{attribute 'qualified_only'}
VAR_GLOBAL
		Device_1_EtherCAT : Device_1_EtherCAT_9EEE92A7;
END_VAR

(* stored: Version 1.2.0.0, ProductVersion 3.1.4024.11
   GVL GVL_iXlinker: Id {c7a45b7d-9f22-4e2b-b89e-542f37f3c2e8} *)
